// TIA Portal project "solar_panel" (V15)

(* hardware
DEVICE "S7-1200 station_1"  S7-1200 Station
   slot 0: "Rack_0"  S7-1200 Rack  Rack  V1.0
   slot 1: "PLC_1"  CPU 1214C DC/DC/DC  6ES7 214-1AG40-0XB0  V4.2
*)

// ===== PLC "PLC_1"  CPU 1214C DC/DC/DC =====

VAR_GLOBAL   // PLC tag table "Default tag table"
   "Clock_Byte" AT %MB80 : Byte;
   "Clock_10Hz" AT %M80.0 : Bool;
   "Clock_5Hz" AT %M80.1 : Bool;
   "Clock_2.5Hz" AT %M80.2 : Bool;
   "Clock_2Hz" AT %M80.3 : Bool;
   "Clock_1.25Hz" AT %M80.4 : Bool;
   "Clock_1Hz" AT %M80.5 : Bool;
   "Clock_0.625Hz" AT %M80.6 : Bool;
   "Clock_0.5Hz" AT %M80.7 : Bool;
   "Tag_18" AT %M20.0 : Bool;
   "Tag_19" AT %M20.1 : Bool;
   "Tag_3" AT %Q0.0 : Bool;
   "Tag_5" AT %MW12 : Int;
   "Error" AT %MW70 : Int;
END_VAR

ORGANIZATION_BLOCK "Main"   // OB1, LAD, ProgramCycle
TITLE = "Main Program Sweep (Cycle)"
{ S7_Optimized_Access := 'TRUE' }
VERSION : 0.1
   VAR_INPUT
      Initial_Call : Bool;   // Initial call of this OB
      Remanence : Bool;   // =True, if remanent data are available
   END_VAR
BEGIN

REGION Network 1
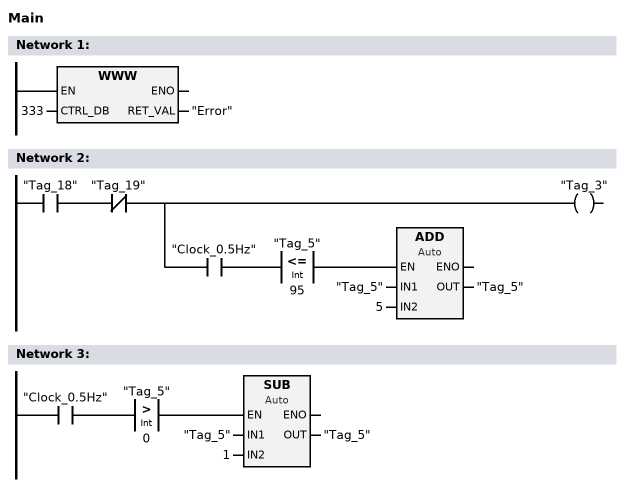
   "Error" := WWW(CTRL_DB := 333);
END_REGION

REGION Network 2
   RUNG wire#powerrail
      Contact( "Tag_18" )
      I_Contact( "Tag_19" )
      wire#w1
      Coil( "Tag_3" )
   END_RUNG
   RUNG wire#w1
      Contact( "Clock_0.5Hz" )
      { S7_Templates := "SrcType := Int" } LE_Contact(in1 := "Tag_5", in2 := 95)
      Add(in1 := "Tag_5", in2 := 5, out => "Tag_5")
   END_RUNG
   // the same network as SCL:
   "Tag_3" := "Tag_18" AND NOT "Tag_19";
   IF "Tag_3" AND "Clock_0.5Hz" AND ("Tag_5" <= 95) THEN "Tag_5" := "Tag_5" + 5; END_IF;
END_REGION

REGION Network 3
   RUNG wire#powerrail
      Contact( "Clock_0.5Hz" )
      { S7_Templates := "SrcType := Int" } GT_Contact(in1 := "Tag_5", in2 := 0)
      Sub(in1 := "Tag_5", in2 := 1, out => "Tag_5")
   END_RUNG
   // the same network as SCL:
   IF "Clock_0.5Hz" AND ("Tag_5" > 0) THEN "Tag_5" := "Tag_5" - 1; END_IF;
END_REGION
END_ORGANIZATION_BLOCK